SUBAPPLICATION DualHysteresis_Thresholds_AR (* Berechnet die 5 Hysterese-Schwellwerte (MID, MID+/-DEAD, MID+/-DEAD+/-HYST) aus MI, DEAD und HYST ueber AR-Adapter; inklusive Durchreich-Plugs MI_OUT, DEAD_OUT und HYST_OUT *)
  (* Standard: 61499-2; Description: Copyright (c) 2026 Meisterschulen am Ostbahnhof This program and the accompanying materials are made available under the terms of the Eclipse Public License 2.0 which is available at https://www.eclipse.org/legal/epl-2.0/ SPDX-License-Identifier: EPL-2.0 *)
  (* Version 1.1, 2026-09-27, Franz Höpfinger, Meisterschulen am Ostbahnhof, MI_OUT Durchreich-Plug ergaenzt (Split_MI zu AR_SPLIT_4), damit MI_OUT und MID_OUT getrennt sind und Adapter nie ohne Split verzweigt werden *)
  (* Version 1.0, 2026-09-27, Franz Höpfinger, Meisterschulen am Ostbahnhof, initial API and implementation *)
  PACKAGE MyLib::sys;
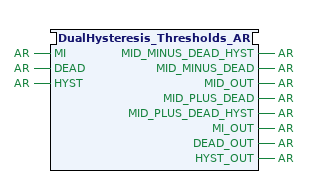
  SOCKETS
    MI : adapter::types::unidirectional::AR; (* Sollwert / Mittelwert (Center Point) *)
    DEAD : adapter::types::unidirectional::AR; (* Totzone um MI (Deadband) *)
    HYST : adapter::types::unidirectional::AR; (* Hysterese zusaetzlich zur Totzone *)
  END_SOCKETS
  PLUGS
    MID_MINUS_DEAD_HYST : adapter::types::unidirectional::AR; (* Schwelle 1: MI - (DEAD + HYST) [Min / Heben Ein / Senken Start] *)
    MID_MINUS_DEAD : adapter::types::unidirectional::AR; (* Schwelle 2: MI - DEAD [Senken Stopp] *)
    MID_OUT : adapter::types::unidirectional::AR; (* Schwelle 3: MI (Mitte / Sollwert) fuer Schwellwert-Marker *)
    MID_PLUS_DEAD : adapter::types::unidirectional::AR; (* Schwelle 4: MI + DEAD [Heben Stopp] *)
    MID_PLUS_DEAD_HYST : adapter::types::unidirectional::AR; (* Schwelle 5: MI + (DEAD + HYST) [Max / Heben Start] *)
    MI_OUT : adapter::types::unidirectional::AR; (* Durchreich-Plug fuer MI (z.B. fuer DualHysteresis_AR_AX) *)
    DEAD_OUT : adapter::types::unidirectional::AR; (* Durchreich-Plug fuer DEAD (z.B. fuer DualHysteresis_AR_AX) *)
    HYST_OUT : adapter::types::unidirectional::AR; (* Durchreich-Plug fuer HYST (z.B. fuer DualHysteresis_AR_AX) *)
  END_PLUGS
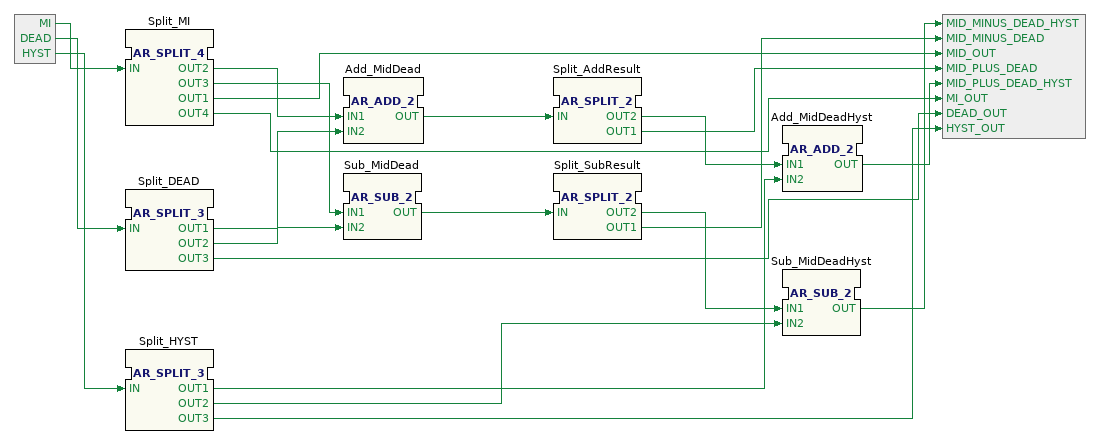
  FBS
    Split_MI : adapter::events::unidirectional::AR_SPLIT_4;
    Split_DEAD : adapter::events::unidirectional::AR_SPLIT_3;
    Split_HYST : adapter::events::unidirectional::AR_SPLIT_3;
    Add_MidDead : adapter::iec61131::arithmetic::AR_ADD_2;
    Sub_MidDead : adapter::iec61131::arithmetic::AR_SUB_2;
    Split_AddResult : adapter::events::unidirectional::AR_SPLIT_2;
    Split_SubResult : adapter::events::unidirectional::AR_SPLIT_2;
    Add_MidDeadHyst : adapter::iec61131::arithmetic::AR_ADD_2;
    Sub_MidDeadHyst : adapter::iec61131::arithmetic::AR_SUB_2;
  END_FBS
  ADAPTER_CONNECTIONS
    MI TO Split_MI.IN;
    DEAD TO Split_DEAD.IN;
    HYST TO Split_HYST.IN;
    Split_MI.OUT2 TO Add_MidDead.IN1;
    Split_DEAD.OUT1 TO Add_MidDead.IN2;
    Split_MI.OUT3 TO Sub_MidDead.IN1;
    Split_DEAD.OUT2 TO Sub_MidDead.IN2;
    Add_MidDead.OUT TO Split_AddResult.IN;
    Sub_MidDead.OUT TO Split_SubResult.IN;
    Split_AddResult.OUT2 TO Add_MidDeadHyst.IN1;
    Split_HYST.OUT1 TO Add_MidDeadHyst.IN2;
    Split_SubResult.OUT2 TO Sub_MidDeadHyst.IN1;
    Split_HYST.OUT2 TO Sub_MidDeadHyst.IN2;
    Split_MI.OUT1 TO MID_OUT;
    Split_AddResult.OUT1 TO MID_PLUS_DEAD;
    Split_SubResult.OUT1 TO MID_MINUS_DEAD;
    Add_MidDeadHyst.OUT TO MID_PLUS_DEAD_HYST;
    Sub_MidDeadHyst.OUT TO MID_MINUS_DEAD_HYST;
    Split_MI.OUT4 TO MI_OUT;
    Split_DEAD.OUT3 TO DEAD_OUT;
    Split_HYST.OUT3 TO HYST_OUT;
  END_CONNECTIONS
END_SUBAPPLICATION
